// TIA Portal V19 export
FUNCTION_BLOCK "F_Zone05_FB"   // FB116, F_LAD
TITLE = SAFETY ZONE 07 - AREA 01 (PEELERS + STRAIGHTENER + JB + LOOP 1 FRONT)
// stored: Access Published
   VAR
      D04 : "Door_FB";
      D05 : "Door_FB";
      FNS : "ForceNormalStop";
      F_SafetyValve_CoilCar : "FDevice_Valve_FB";
      F_SafetyValve_Peeler : "FDevice_Valve_FB";
      F_SafetyValve_JB_Cut_Rest : "FDevice_Valve_FB";
      F_SafetyValve_JB_Cut_Work : "FDevice_Valve_FB";
      F_Contactor_HU_Area01_Motor : "FDevice_Contactor_FB";
      F_Sinamics_JBTorch : "FDevice_Sinamics_FB";
      F_Sinamics_JBPinchRoll : "FDevice_Sinamics_FB";
   END_VAR
   VAR_TEMP
      Fdbk : Bool;
   END_VAR
   VAR CONSTANT
      JB_TORCH_S120_STOPPING_TIME : Time := T#1s;
      JB_PINCHR_S120_STOPPING_TIME : Time := T#1s;
   END_VAR
BEGIN

REGION Network 1: < < < < < < < < < < DOOR > > > > > > > > > >
END_REGION

REGION Network 2: Zone Entry enable
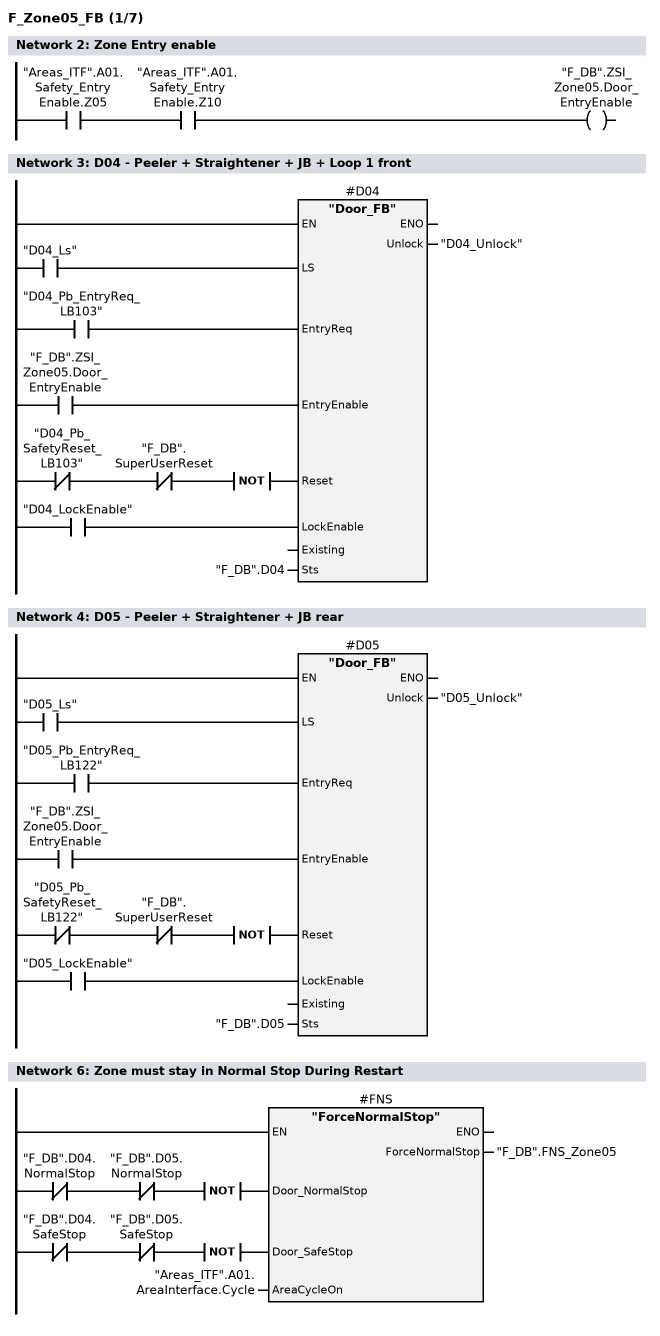
   RUNG wire#powerrail
      Contact( "Areas_ITF".A01.Safety_EntryEnable.Z05 )
      Contact( "Areas_ITF".A01.Safety_EntryEnable.Z10 )
      Coil( "F_DB".ZSI_Zone05.Door_EntryEnable )
   END_RUNG
   // the same network as SCL:
   "F_DB".ZSI_Zone05.Door_EntryEnable := "Areas_ITF".A01.Safety_EntryEnable.Z05 AND "Areas_ITF".A01.Safety_EntryEnable.Z10;
END_REGION

REGION Network 3: D04 - Peeler + Straightener + JB + Loop 1 front
   RUNG wire#powerrail
      #D04(LS := wire#w1, EntryReq := wire#w2, EntryEnable := wire#w3, Reset := wire#w4, LockEnable := wire#w5, Existing :=, Sts := "F_DB".D04, Unlock => "D04_Unlock")
   END_RUNG
   RUNG wire#powerrail
      Contact( "D04_Ls" )
   END_RUNG wire#w1
   RUNG wire#powerrail
      Contact( "D04_Pb_EntryReq_LB103" )
   END_RUNG wire#w2
   RUNG wire#powerrail
      Contact( "F_DB".ZSI_Zone05.Door_EntryEnable )
   END_RUNG wire#w3
   RUNG wire#powerrail
      I_Contact( "D04_Pb_SafetyReset_LB103" )
      I_Contact( "F_DB".SuperUserReset )
      Not()
   END_RUNG wire#w4
   RUNG wire#powerrail
      Contact( "D04_LockEnable" )
   END_RUNG wire#w5
   // the same network as SCL:
   #D04(LS := "D04_Ls",   // "Door_FB"
        EntryReq := "D04_Pb_EntryReq_LB103",
        EntryEnable := "F_DB".ZSI_Zone05.Door_EntryEnable,
        Reset := NOT (NOT "D04_Pb_SafetyReset_LB103" AND NOT "F_DB".SuperUserReset),
        LockEnable := "D04_LockEnable",
        Sts := "F_DB".D04,
        Unlock => "D04_Unlock");
END_REGION

REGION Network 4: D05 - Peeler + Straightener + JB rear
   RUNG wire#powerrail
      #D05(LS := wire#w1, EntryReq := wire#w2, EntryEnable := wire#w3, Reset := wire#w4, LockEnable := wire#w5, Existing :=, Sts := "F_DB".D05, Unlock => "D05_Unlock")
   END_RUNG
   RUNG wire#powerrail
      Contact( "D05_Ls" )
   END_RUNG wire#w1
   RUNG wire#powerrail
      Contact( "D05_Pb_EntryReq_LB122" )
   END_RUNG wire#w2
   RUNG wire#powerrail
      Contact( "F_DB".ZSI_Zone05.Door_EntryEnable )
   END_RUNG wire#w3
   RUNG wire#powerrail
      I_Contact( "D05_Pb_SafetyReset_LB122" )
      I_Contact( "F_DB".SuperUserReset )
      Not()
   END_RUNG wire#w4
   RUNG wire#powerrail
      Contact( "D05_LockEnable" )
   END_RUNG wire#w5
   // the same network as SCL:
   #D05(LS := "D05_Ls",   // "Door_FB"
        EntryReq := "D05_Pb_EntryReq_LB122",
        EntryEnable := "F_DB".ZSI_Zone05.Door_EntryEnable,
        Reset := NOT (NOT "D05_Pb_SafetyReset_LB122" AND NOT "F_DB".SuperUserReset),
        LockEnable := "D05_LockEnable",
        Sts := "F_DB".D05,
        Unlock => "D05_Unlock");
END_REGION

REGION Network 5: < < < < < < < < < < FORCE NORMAL STOP > > > > > > > > > >
END_REGION

REGION Network 6: Zone must stay in Normal Stop During Restart
   RUNG wire#powerrail
      #FNS(Door_NormalStop := wire#w1, Door_SafeStop := wire#w2, AreaCycleOn := "Areas_ITF".A01.AreaInterface.Cycle, ForceNormalStop => "F_DB".FNS_Zone05)
   END_RUNG
   RUNG wire#powerrail
      I_Contact( "F_DB".D04.NormalStop )
      I_Contact( "F_DB".D05.NormalStop )
      Not()
   END_RUNG wire#w1
   RUNG wire#powerrail
      I_Contact( "F_DB".D04.SafeStop )
      I_Contact( "F_DB".D05.SafeStop )
      Not()
   END_RUNG wire#w2
   // the same network as SCL:
   #FNS(Door_NormalStop := NOT (NOT "F_DB".D04.NormalStop AND NOT "F_DB".D05.NormalStop),   // "ForceNormalStop"
        Door_SafeStop := NOT (NOT "F_DB".D04.SafeStop AND NOT "F_DB".D05.SafeStop),
        AreaCycleOn := "Areas_ITF".A01.AreaInterface.Cycle,
        ForceNormalStop => "F_DB".FNS_Zone05);
END_REGION

REGION Network 7: < < < < < < < < < < ZONE SAFETY INTERFACE > > > > > > > > > >
END_REGION

REGION Network 8: Cumulative Zone Safety
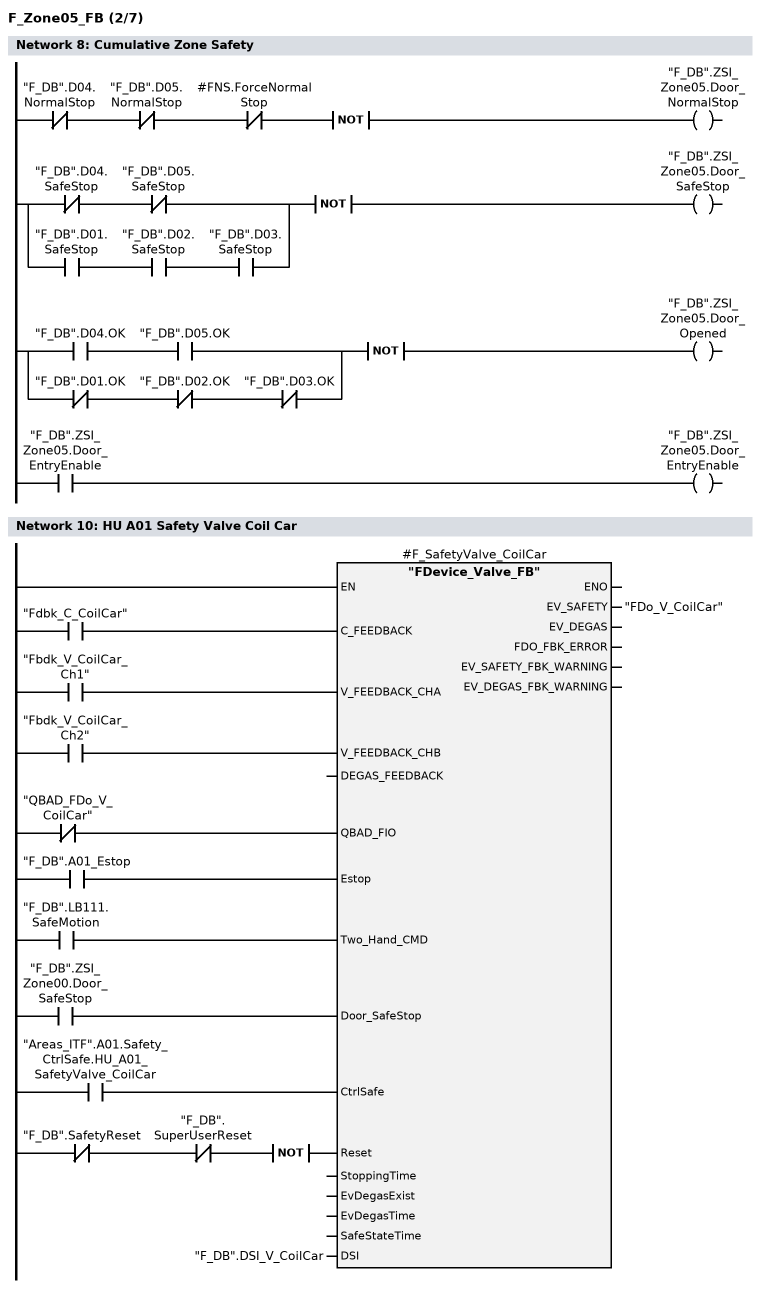
   RUNG wire#powerrail
      I_Contact( "F_DB".D04.NormalStop )
      I_Contact( "F_DB".D05.NormalStop )
      I_Contact( #FNS.ForceNormalStop )
      Not()
      Coil( "F_DB".ZSI_Zone05.Door_NormalStop )
   END_RUNG
   RUNG wire#powerrail
      I_Contact( "F_DB".D04.SafeStop )
      I_Contact( "F_DB".D05.SafeStop )
      wire#w1
      Not()
      Coil( "F_DB".ZSI_Zone05.Door_SafeStop )
   END_RUNG
   RUNG wire#powerrail
      Contact( "F_DB".D01.SafeStop )
      Contact( "F_DB".D02.SafeStop )
      Contact( "F_DB".D03.SafeStop )
   END_RUNG wire#w1
   RUNG wire#powerrail
      Contact( "F_DB".D04.OK )
      Contact( "F_DB".D05.OK )
      wire#w2
      Not()
      Coil( "F_DB".ZSI_Zone05.Door_Opened )
   END_RUNG
   RUNG wire#powerrail
      I_Contact( "F_DB".D01.OK )
      I_Contact( "F_DB".D02.OK )
      I_Contact( "F_DB".D03.OK )
   END_RUNG wire#w2
   RUNG wire#powerrail
      Contact( "F_DB".ZSI_Zone05.Door_EntryEnable )
      Coil( "F_DB".ZSI_Zone05.Door_EntryEnable )
   END_RUNG
   // the same network as SCL:
   "F_DB".ZSI_Zone05.Door_NormalStop := NOT (NOT "F_DB".D04.NormalStop AND NOT "F_DB".D05.NormalStop AND NOT #FNS.ForceNormalStop);
   "F_DB".ZSI_Zone05.Door_SafeStop := NOT ((NOT "F_DB".D04.SafeStop AND NOT "F_DB".D05.SafeStop) OR ("F_DB".D01.SafeStop AND "F_DB".D02.SafeStop AND "F_DB".D03.SafeStop));
   "F_DB".ZSI_Zone05.Door_Opened := NOT (("F_DB".D04.OK AND "F_DB".D05.OK) OR (NOT "F_DB".D01.OK AND NOT "F_DB".D02.OK AND NOT "F_DB".D03.OK));
   "F_DB".ZSI_Zone05.Door_EntryEnable := "F_DB".ZSI_Zone05.Door_EntryEnable;
END_REGION

REGION Network 9: < < < < < < < < < < DEVICES SAFETY VALVES > > > > > > > > > >
END_REGION

REGION Network 10: HU A01 Safety Valve Coil Car
   RUNG wire#powerrail
      #F_SafetyValve_CoilCar(C_FEEDBACK := wire#w1, V_FEEDBACK_CHA := wire#w2, V_FEEDBACK_CHB := wire#w3, QBAD_FIO := wire#w4, Estop := wire#w5, Two_Hand_CMD := wire#w6, Door_SafeStop := wire#w7, CtrlSafe := wire#w8, Reset := wire#w9, DEGAS_FEEDBACK :=, StoppingTime :=, EvDegasExist :=, EvDegasTime :=, SafeStateTime :=, DSI := "F_DB".DSI_V_CoilCar, EV_SAFETY => "FDo_V_CoilCar", EV_DEGAS =>, FDO_FBK_ERROR =>, EV_SAFETY_FBK_WARNING =>, EV_DEGAS_FBK_WARNING =>)
   END_RUNG
   RUNG wire#powerrail
      Contact( "Fdbk_C_CoilCar" )
   END_RUNG wire#w1
   RUNG wire#powerrail
      Contact( "Fbdk_V_CoilCar_Ch1" )
   END_RUNG wire#w2
   RUNG wire#powerrail
      Contact( "Fbdk_V_CoilCar_Ch2" )
   END_RUNG wire#w3
   RUNG wire#powerrail
      I_Contact( "QBAD_FDo_V_CoilCar" )
   END_RUNG wire#w4
   RUNG wire#powerrail
      Contact( "F_DB".A01_Estop )
   END_RUNG wire#w5
   RUNG wire#powerrail
      Contact( "F_DB".LB111.SafeMotion )
   END_RUNG wire#w6
   RUNG wire#powerrail
      Contact( "F_DB".ZSI_Zone00.Door_SafeStop )
   END_RUNG wire#w7
   RUNG wire#powerrail
      Contact( "Areas_ITF".A01.Safety_CtrlSafe.HU_A01_SafetyValve_CoilCar )
   END_RUNG wire#w8
   RUNG wire#powerrail
      I_Contact( "F_DB".SafetyReset )
      I_Contact( "F_DB".SuperUserReset )
      Not()
   END_RUNG wire#w9
   // the same network as SCL:
   #F_SafetyValve_CoilCar(C_FEEDBACK := "Fdbk_C_CoilCar",   // "FDevice_Valve_FB"
                          V_FEEDBACK_CHA := "Fbdk_V_CoilCar_Ch1",
                          V_FEEDBACK_CHB := "Fbdk_V_CoilCar_Ch2",
                          QBAD_FIO := NOT "QBAD_FDo_V_CoilCar",
                          Estop := "F_DB".A01_Estop,
                          Two_Hand_CMD := "F_DB".LB111.SafeMotion,
                          Door_SafeStop := "F_DB".ZSI_Zone00.Door_SafeStop,
                          CtrlSafe := "Areas_ITF".A01.Safety_CtrlSafe.HU_A01_SafetyValve_CoilCar,
                          Reset := NOT (NOT "F_DB".SafetyReset AND NOT "F_DB".SuperUserReset),
                          DSI := "F_DB".DSI_V_CoilCar,
                          EV_SAFETY => "FDo_V_CoilCar");
END_REGION

REGION Network 11: HU A01 Safety Valve Peeler
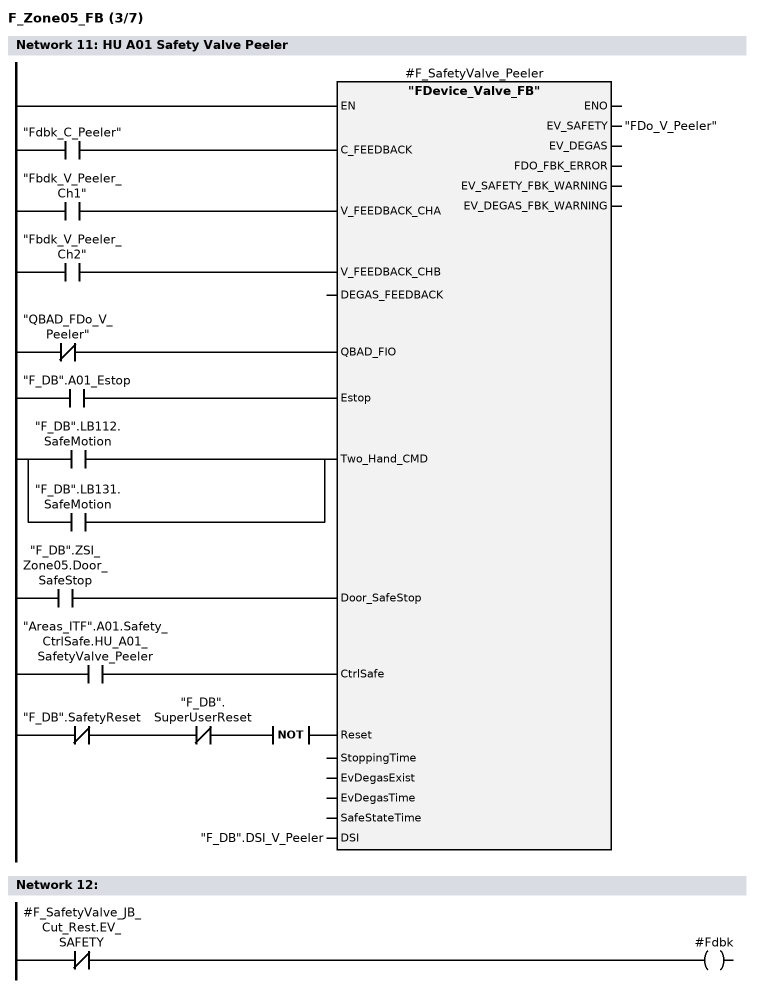
   RUNG wire#powerrail
      #F_SafetyValve_Peeler(C_FEEDBACK := wire#w1, V_FEEDBACK_CHA := wire#w2, V_FEEDBACK_CHB := wire#w3, QBAD_FIO := wire#w4, Estop := wire#w5, Two_Hand_CMD := wire#w6, Door_SafeStop := wire#w7, CtrlSafe := wire#w8, Reset := wire#w9, DEGAS_FEEDBACK :=, StoppingTime :=, EvDegasExist :=, EvDegasTime :=, SafeStateTime :=, DSI := "F_DB".DSI_V_Peeler, EV_SAFETY => "FDo_V_Peeler", EV_DEGAS =>, FDO_FBK_ERROR =>, EV_SAFETY_FBK_WARNING =>, EV_DEGAS_FBK_WARNING =>)
   END_RUNG
   RUNG wire#powerrail
      Contact( "Fdbk_C_Peeler" )
   END_RUNG wire#w1
   RUNG wire#powerrail
      Contact( "Fbdk_V_Peeler_Ch1" )
   END_RUNG wire#w2
   RUNG wire#powerrail
      Contact( "Fbdk_V_Peeler_Ch2" )
   END_RUNG wire#w3
   RUNG wire#powerrail
      I_Contact( "QBAD_FDo_V_Peeler" )
   END_RUNG wire#w4
   RUNG wire#powerrail
      Contact( "F_DB".A01_Estop )
   END_RUNG wire#w5
   RUNG wire#powerrail
      Contact( "F_DB".LB112.SafeMotion )
   END_RUNG wire#w6
   RUNG wire#powerrail
      Contact( "F_DB".LB131.SafeMotion )
   END_RUNG wire#w6
   RUNG wire#powerrail
      Contact( "F_DB".ZSI_Zone05.Door_SafeStop )
   END_RUNG wire#w7
   RUNG wire#powerrail
      Contact( "Areas_ITF".A01.Safety_CtrlSafe.HU_A01_SafetyValve_Peeler )
   END_RUNG wire#w8
   RUNG wire#powerrail
      I_Contact( "F_DB".SafetyReset )
      I_Contact( "F_DB".SuperUserReset )
      Not()
   END_RUNG wire#w9
   // the same network as SCL:
   #F_SafetyValve_Peeler(C_FEEDBACK := "Fdbk_C_Peeler",   // "FDevice_Valve_FB"
                         V_FEEDBACK_CHA := "Fbdk_V_Peeler_Ch1",
                         V_FEEDBACK_CHB := "Fbdk_V_Peeler_Ch2",
                         QBAD_FIO := NOT "QBAD_FDo_V_Peeler",
                         Estop := "F_DB".A01_Estop,
                         Two_Hand_CMD := "F_DB".LB112.SafeMotion OR "F_DB".LB131.SafeMotion,
                         Door_SafeStop := "F_DB".ZSI_Zone05.Door_SafeStop,
                         CtrlSafe := "Areas_ITF".A01.Safety_CtrlSafe.HU_A01_SafetyValve_Peeler,
                         Reset := NOT (NOT "F_DB".SafetyReset AND NOT "F_DB".SuperUserReset),
                         DSI := "F_DB".DSI_V_Peeler,
                         EV_SAFETY => "FDo_V_Peeler");
END_REGION

REGION Network 12
   RUNG wire#powerrail
      I_Contact( #F_SafetyValve_JB_Cut_Rest.EV_SAFETY )
      Coil( #Fdbk )
   END_RUNG
   // the same network as SCL:
   #Fdbk := NOT #F_SafetyValve_JB_Cut_Rest.EV_SAFETY;
END_REGION

REGION Network 13: HU A01 Safety Valve JB Cut Rest
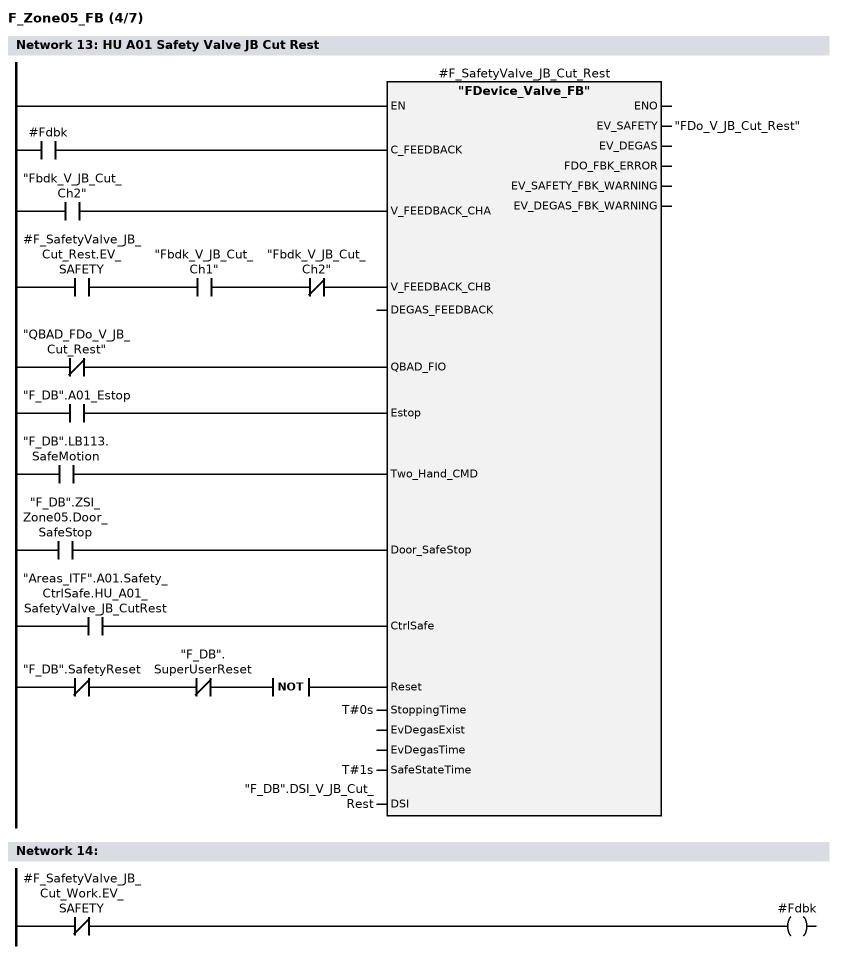
   RUNG wire#powerrail
      #F_SafetyValve_JB_Cut_Rest(C_FEEDBACK := wire#w1, V_FEEDBACK_CHA := wire#w2, V_FEEDBACK_CHB := wire#w3, QBAD_FIO := wire#w4, Estop := wire#w5, Two_Hand_CMD := wire#w6, Door_SafeStop := wire#w7, CtrlSafe := wire#w8, Reset := wire#w9, DEGAS_FEEDBACK :=, StoppingTime := T#0s, EvDegasExist :=, EvDegasTime :=, SafeStateTime := T#1s, DSI := "F_DB".DSI_V_JB_Cut_Rest, EV_SAFETY => "FDo_V_JB_Cut_Rest", EV_DEGAS =>, FDO_FBK_ERROR =>, EV_SAFETY_FBK_WARNING =>, EV_DEGAS_FBK_WARNING =>)
   END_RUNG
   RUNG wire#powerrail
      Contact( #Fdbk )
   END_RUNG wire#w1
   RUNG wire#powerrail
      Contact( "Fbdk_V_JB_Cut_Ch2" )
   END_RUNG wire#w2
   RUNG wire#powerrail
      Contact( #F_SafetyValve_JB_Cut_Rest.EV_SAFETY )
      Contact( "Fbdk_V_JB_Cut_Ch1" )
      I_Contact( "Fbdk_V_JB_Cut_Ch2" )
   END_RUNG wire#w3
   RUNG wire#powerrail
      I_Contact( "QBAD_FDo_V_JB_Cut_Rest" )
   END_RUNG wire#w4
   RUNG wire#powerrail
      Contact( "F_DB".A01_Estop )
   END_RUNG wire#w5
   RUNG wire#powerrail
      Contact( "F_DB".LB113.SafeMotion )
   END_RUNG wire#w6
   RUNG wire#powerrail
      Contact( "F_DB".ZSI_Zone05.Door_SafeStop )
   END_RUNG wire#w7
   RUNG wire#powerrail
      Contact( "Areas_ITF".A01.Safety_CtrlSafe.HU_A01_SafetyValve_JB_CutRest )
   END_RUNG wire#w8
   RUNG wire#powerrail
      I_Contact( "F_DB".SafetyReset )
      I_Contact( "F_DB".SuperUserReset )
      Not()
   END_RUNG wire#w9
   // the same network as SCL:
   #F_SafetyValve_JB_Cut_Rest(C_FEEDBACK := #Fdbk,   // "FDevice_Valve_FB"
                           V_FEEDBACK_CHA := "Fbdk_V_JB_Cut_Ch2",
                           V_FEEDBACK_CHB := #F_SafetyValve_JB_Cut_Rest.EV_SAFETY AND "Fbdk_V_JB_Cut_Ch1" AND NOT "Fbdk_V_JB_Cut_Ch2",
                           QBAD_FIO := NOT "QBAD_FDo_V_JB_Cut_Rest",
                           Estop := "F_DB".A01_Estop,
                           Two_Hand_CMD := "F_DB".LB113.SafeMotion,
                           Door_SafeStop := "F_DB".ZSI_Zone05.Door_SafeStop,
                           CtrlSafe := "Areas_ITF".A01.Safety_CtrlSafe.HU_A01_SafetyValve_JB_CutRest,
                           Reset := NOT (NOT "F_DB".SafetyReset AND NOT "F_DB".SuperUserReset),
                           StoppingTime := T#0s,
                           SafeStateTime := T#1s,
                           DSI := "F_DB".DSI_V_JB_Cut_Rest,
                           EV_SAFETY => "FDo_V_JB_Cut_Rest");
END_REGION

REGION Network 14
   RUNG wire#powerrail
      I_Contact( #F_SafetyValve_JB_Cut_Work.EV_SAFETY )
      Coil( #Fdbk )
   END_RUNG
   // the same network as SCL:
   #Fdbk := NOT #F_SafetyValve_JB_Cut_Work.EV_SAFETY;
END_REGION

REGION Network 15: HU A01 Safety Valve JB Cut Work
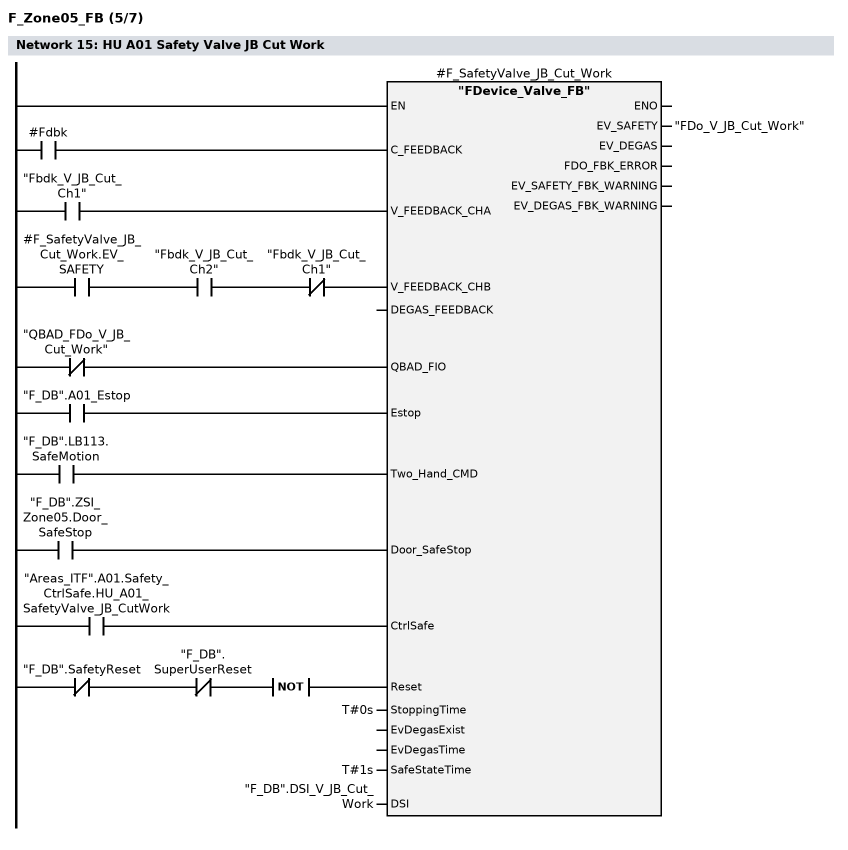
   RUNG wire#powerrail
      #F_SafetyValve_JB_Cut_Work(C_FEEDBACK := wire#w1, V_FEEDBACK_CHA := wire#w2, V_FEEDBACK_CHB := wire#w3, QBAD_FIO := wire#w4, Estop := wire#w5, Two_Hand_CMD := wire#w6, Door_SafeStop := wire#w7, CtrlSafe := wire#w8, Reset := wire#w9, DEGAS_FEEDBACK :=, StoppingTime := T#0s, EvDegasExist :=, EvDegasTime :=, SafeStateTime := T#1s, DSI := "F_DB".DSI_V_JB_Cut_Work, EV_SAFETY => "FDo_V_JB_Cut_Work", EV_DEGAS =>, FDO_FBK_ERROR =>, EV_SAFETY_FBK_WARNING =>, EV_DEGAS_FBK_WARNING =>)
   END_RUNG
   RUNG wire#powerrail
      Contact( #Fdbk )
   END_RUNG wire#w1
   RUNG wire#powerrail
      Contact( "Fbdk_V_JB_Cut_Ch1" )
   END_RUNG wire#w2
   RUNG wire#powerrail
      Contact( #F_SafetyValve_JB_Cut_Work.EV_SAFETY )
      Contact( "Fbdk_V_JB_Cut_Ch2" )
      I_Contact( "Fbdk_V_JB_Cut_Ch1" )
   END_RUNG wire#w3
   RUNG wire#powerrail
      I_Contact( "QBAD_FDo_V_JB_Cut_Work" )
   END_RUNG wire#w4
   RUNG wire#powerrail
      Contact( "F_DB".A01_Estop )
   END_RUNG wire#w5
   RUNG wire#powerrail
      Contact( "F_DB".LB113.SafeMotion )
   END_RUNG wire#w6
   RUNG wire#powerrail
      Contact( "F_DB".ZSI_Zone05.Door_SafeStop )
   END_RUNG wire#w7
   RUNG wire#powerrail
      Contact( "Areas_ITF".A01.Safety_CtrlSafe.HU_A01_SafetyValve_JB_CutWork )
   END_RUNG wire#w8
   RUNG wire#powerrail
      I_Contact( "F_DB".SafetyReset )
      I_Contact( "F_DB".SuperUserReset )
      Not()
   END_RUNG wire#w9
   // the same network as SCL:
   #F_SafetyValve_JB_Cut_Work(C_FEEDBACK := #Fdbk,   // "FDevice_Valve_FB"
                           V_FEEDBACK_CHA := "Fbdk_V_JB_Cut_Ch1",
                           V_FEEDBACK_CHB := #F_SafetyValve_JB_Cut_Work.EV_SAFETY AND "Fbdk_V_JB_Cut_Ch2" AND NOT "Fbdk_V_JB_Cut_Ch1",
                           QBAD_FIO := NOT "QBAD_FDo_V_JB_Cut_Work",
                           Estop := "F_DB".A01_Estop,
                           Two_Hand_CMD := "F_DB".LB113.SafeMotion,
                           Door_SafeStop := "F_DB".ZSI_Zone05.Door_SafeStop,
                           CtrlSafe := "Areas_ITF".A01.Safety_CtrlSafe.HU_A01_SafetyValve_JB_CutWork,
                           Reset := NOT (NOT "F_DB".SafetyReset AND NOT "F_DB".SuperUserReset),
                           StoppingTime := T#0s,
                           SafeStateTime := T#1s,
                           DSI := "F_DB".DSI_V_JB_Cut_Work,
                           EV_SAFETY => "FDo_V_JB_Cut_Work");
END_REGION

REGION Network 16: >
END_REGION

REGION Network 17: < < < < < < < < < < DEVICES CONTACTORS > > > > > > > > > >
END_REGION

REGION Network 18: HU A01 Motor contactor
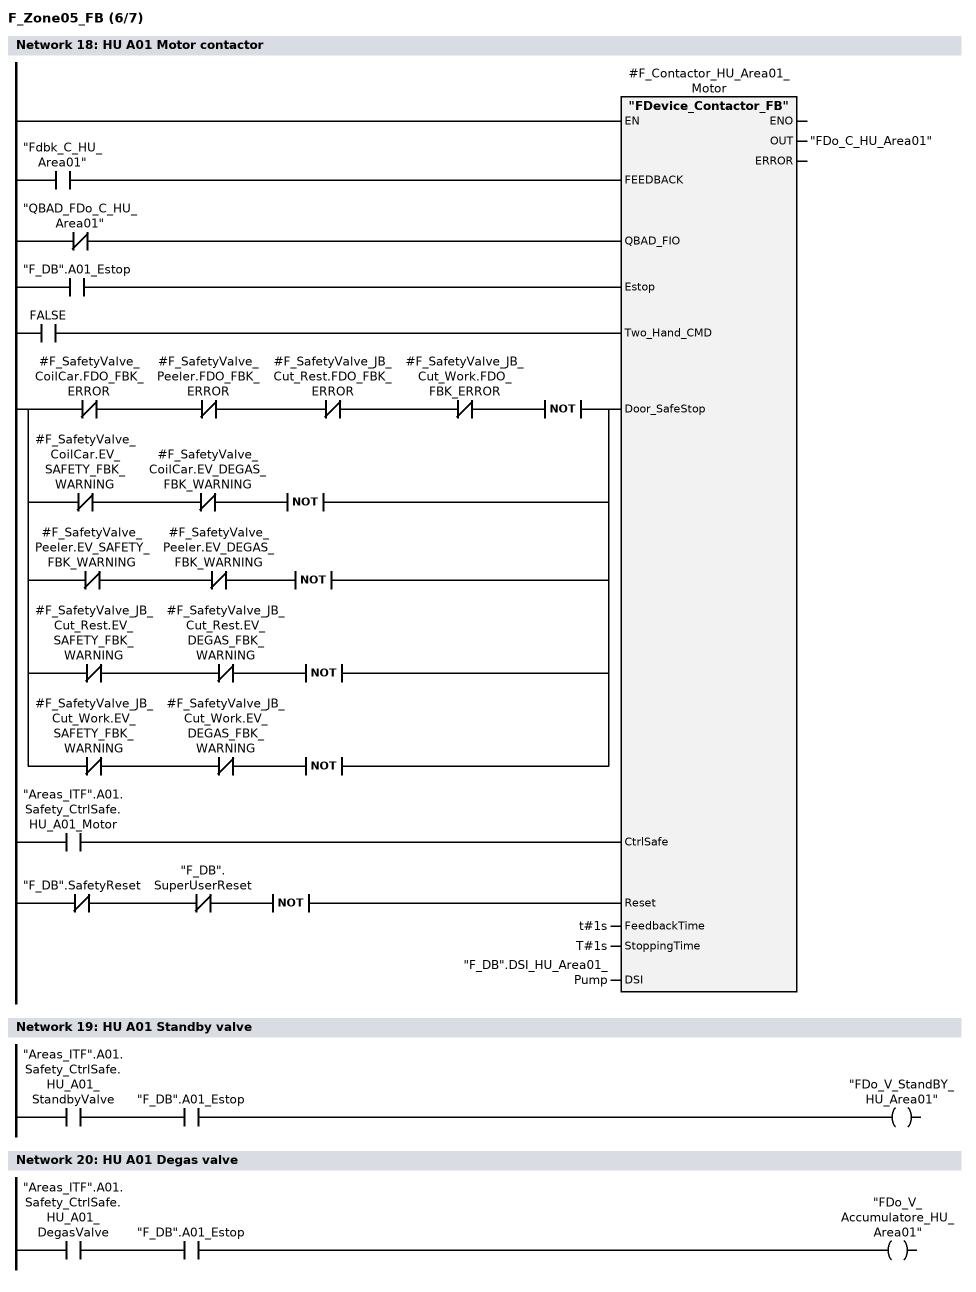
   RUNG wire#powerrail
      #F_Contactor_HU_Area01_Motor(FEEDBACK := wire#w1, QBAD_FIO := wire#w2, Estop := wire#w3, Two_Hand_CMD := wire#w4, Door_SafeStop := wire#w5, CtrlSafe := wire#w6, Reset := wire#w7, FeedbackTime := t#1s, StoppingTime := T#1s, DSI := "F_DB".DSI_HU_Area01_Pump, OUT => "FDo_C_HU_Area01", ERROR =>)
   END_RUNG
   RUNG wire#powerrail
      Contact( "Fdbk_C_HU_Area01" )
   END_RUNG wire#w1
   RUNG wire#powerrail
      I_Contact( "QBAD_FDo_C_HU_Area01" )
   END_RUNG wire#w2
   RUNG wire#powerrail
      Contact( "F_DB".A01_Estop )
   END_RUNG wire#w3
   RUNG wire#powerrail
      Contact( FALSE )
   END_RUNG wire#w4
   RUNG wire#powerrail
      I_Contact( #F_SafetyValve_CoilCar.FDO_FBK_ERROR )
      I_Contact( #F_SafetyValve_Peeler.FDO_FBK_ERROR )
      I_Contact( #F_SafetyValve_JB_Cut_Rest.FDO_FBK_ERROR )
      I_Contact( #F_SafetyValve_JB_Cut_Work.FDO_FBK_ERROR )
      Not()
   END_RUNG wire#w5
   RUNG wire#powerrail
      I_Contact( #F_SafetyValve_CoilCar.EV_SAFETY_FBK_WARNING )
      I_Contact( #F_SafetyValve_CoilCar.EV_DEGAS_FBK_WARNING )
      Not()
   END_RUNG wire#w5
   RUNG wire#powerrail
      I_Contact( #F_SafetyValve_Peeler.EV_SAFETY_FBK_WARNING )
      I_Contact( #F_SafetyValve_Peeler.EV_DEGAS_FBK_WARNING )
      Not()
   END_RUNG wire#w5
   RUNG wire#powerrail
      I_Contact( #F_SafetyValve_JB_Cut_Rest.EV_SAFETY_FBK_WARNING )
      I_Contact( #F_SafetyValve_JB_Cut_Rest.EV_DEGAS_FBK_WARNING )
      Not()
   END_RUNG wire#w5
   RUNG wire#powerrail
      I_Contact( #F_SafetyValve_JB_Cut_Work.EV_SAFETY_FBK_WARNING )
      I_Contact( #F_SafetyValve_JB_Cut_Work.EV_DEGAS_FBK_WARNING )
      Not()
   END_RUNG wire#w5
   RUNG wire#powerrail
      Contact( "Areas_ITF".A01.Safety_CtrlSafe.HU_A01_Motor )
   END_RUNG wire#w6
   RUNG wire#powerrail
      I_Contact( "F_DB".SafetyReset )
      I_Contact( "F_DB".SuperUserReset )
      Not()
   END_RUNG wire#w7
   // the same network as SCL:
   #F_Contactor_HU_Area01_Motor(FEEDBACK := "Fdbk_C_HU_Area01",   // "FDevice_Contactor_FB"
                           QBAD_FIO := NOT "QBAD_FDo_C_HU_Area01",
                           Estop := "F_DB".A01_Estop,
                           Two_Hand_CMD := FALSE,
                           Door_SafeStop := NOT (NOT #F_SafetyValve_CoilCar.FDO_FBK_ERROR AND NOT #F_SafetyValve_Peeler.FDO_FBK_ERROR AND NOT #F_SafetyValve_JB_Cut_Rest.FDO_FBK_ERROR AND NOT #F_SafetyValve_JB_Cut_Work.FDO_FBK_ERROR) OR NOT (NOT #F_SafetyValve_CoilCar.EV_SAFETY_FBK_WARNING AND NOT #F_SafetyValve_CoilCar.EV_DEGAS_FBK_WARNING) OR NOT (NOT #F_SafetyValve_Peeler.EV_SAFETY_FBK_WARNING AND NOT #F_SafetyValve_Peeler.EV_DEGAS_FBK_WARNING) OR NOT (NOT #F_SafetyValve_JB_Cut_Rest.EV_SAFETY_FBK_WARNING AND NOT #F_SafetyValve_JB_Cut_Rest.EV_DEGAS_FBK_WARNING) OR NOT (NOT #F_SafetyValve_JB_Cut_Work.EV_SAFETY_FBK_WARNING AND NOT #F_SafetyValve_JB_Cut_Work.EV_DEGAS_FBK_WARNING),
                           CtrlSafe := "Areas_ITF".A01.Safety_CtrlSafe.HU_A01_Motor,
                           Reset := NOT (NOT "F_DB".SafetyReset AND NOT "F_DB".SuperUserReset),
                           FeedbackTime := t#1s,
                           StoppingTime := T#1s,
                           DSI := "F_DB".DSI_HU_Area01_Pump,
                           OUT => "FDo_C_HU_Area01");
END_REGION

REGION Network 19: HU A01 Standby valve
   RUNG wire#powerrail
      Contact( "Areas_ITF".A01.Safety_CtrlSafe.HU_A01_StandbyValve )
      Contact( "F_DB".A01_Estop )
      Coil( "FDo_V_StandBY_HU_Area01" )
   END_RUNG
   // the same network as SCL:
   "FDo_V_StandBY_HU_Area01" := "Areas_ITF".A01.Safety_CtrlSafe.HU_A01_StandbyValve AND "F_DB".A01_Estop;
END_REGION

REGION Network 20: HU A01 Degas valve
   RUNG wire#powerrail
      Contact( "Areas_ITF".A01.Safety_CtrlSafe.HU_A01_DegasValve )
      Contact( "F_DB".A01_Estop )
      Coil( "FDo_V_Accumulatore_HU_Area01" )
   END_RUNG
   // the same network as SCL:
   "FDo_V_Accumulatore_HU_Area01" := "Areas_ITF".A01.Safety_CtrlSafe.HU_A01_DegasValve AND "F_DB".A01_Estop;
END_REGION

REGION Network 21: >
END_REGION

REGION Network 22: < < < < < < < < < < DEVICES S120 > > > > > > > > > >
END_REGION

REGION Network 23: S120 - JB Welder Torch
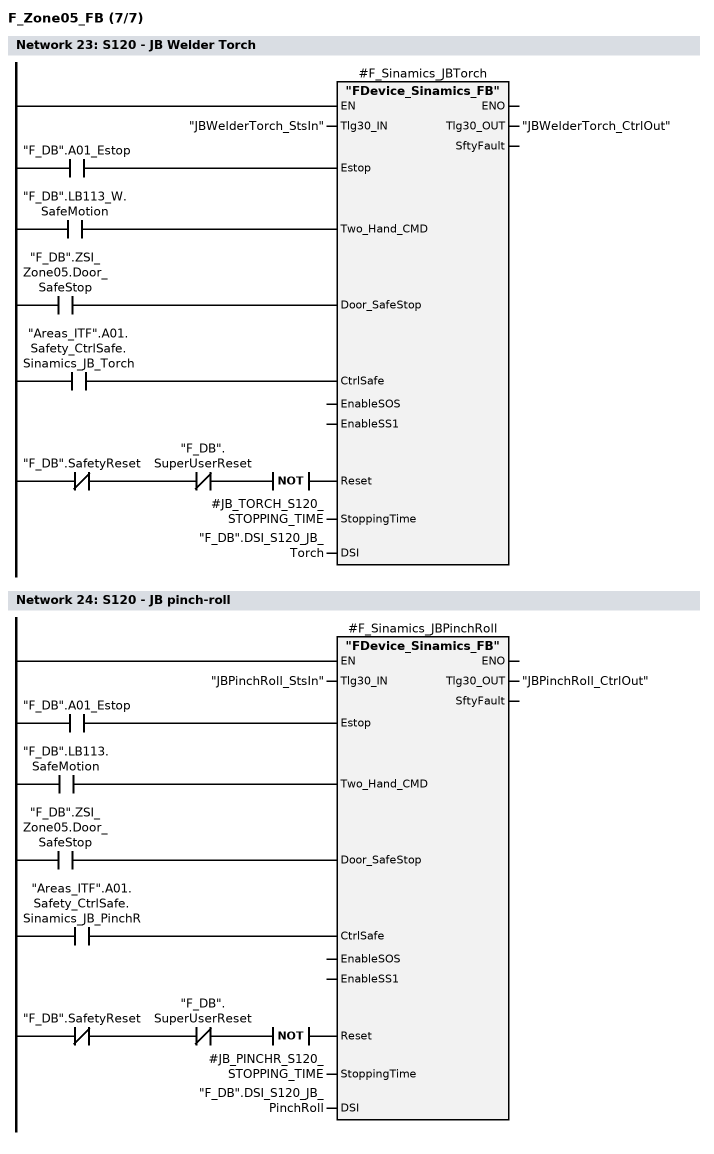
   RUNG wire#powerrail
      #F_Sinamics_JBTorch(Estop := wire#w1, Two_Hand_CMD := wire#w2, Door_SafeStop := wire#w3, CtrlSafe := wire#w4, Reset := wire#w5, Tlg30_IN := "JBWelderTorch_StsIn", EnableSOS :=, EnableSS1 :=, StoppingTime := #JB_TORCH_S120_STOPPING_TIME, DSI := "F_DB".DSI_S120_JB_Torch, Tlg30_OUT => "JBWelderTorch_CtrlOut", SftyFault =>)
   END_RUNG
   RUNG wire#powerrail
      Contact( "F_DB".A01_Estop )
   END_RUNG wire#w1
   RUNG wire#powerrail
      Contact( "F_DB".LB113_W.SafeMotion )
   END_RUNG wire#w2
   RUNG wire#powerrail
      Contact( "F_DB".ZSI_Zone05.Door_SafeStop )
   END_RUNG wire#w3
   RUNG wire#powerrail
      Contact( "Areas_ITF".A01.Safety_CtrlSafe.Sinamics_JB_Torch )
   END_RUNG wire#w4
   RUNG wire#powerrail
      I_Contact( "F_DB".SafetyReset )
      I_Contact( "F_DB".SuperUserReset )
      Not()
   END_RUNG wire#w5
   // the same network as SCL:
   #F_Sinamics_JBTorch(Tlg30_IN := "JBWelderTorch_StsIn",   // "FDevice_Sinamics_FB"
                       Estop := "F_DB".A01_Estop,
                       Two_Hand_CMD := "F_DB".LB113_W.SafeMotion,
                       Door_SafeStop := "F_DB".ZSI_Zone05.Door_SafeStop,
                       CtrlSafe := "Areas_ITF".A01.Safety_CtrlSafe.Sinamics_JB_Torch,
                       Reset := NOT (NOT "F_DB".SafetyReset AND NOT "F_DB".SuperUserReset),
                       StoppingTime := #JB_TORCH_S120_STOPPING_TIME,
                       DSI := "F_DB".DSI_S120_JB_Torch,
                       Tlg30_OUT => "JBWelderTorch_CtrlOut");
END_REGION

REGION Network 24: S120 - JB pinch-roll
   RUNG wire#powerrail
      #F_Sinamics_JBPinchRoll(Estop := wire#w1, Two_Hand_CMD := wire#w2, Door_SafeStop := wire#w3, CtrlSafe := wire#w4, Reset := wire#w5, Tlg30_IN := "JBPinchRoll_StsIn", EnableSOS :=, EnableSS1 :=, StoppingTime := #JB_PINCHR_S120_STOPPING_TIME, DSI := "F_DB".DSI_S120_JB_PinchRoll, Tlg30_OUT => "JBPinchRoll_CtrlOut", SftyFault =>)
   END_RUNG
   RUNG wire#powerrail
      Contact( "F_DB".A01_Estop )
   END_RUNG wire#w1
   RUNG wire#powerrail
      Contact( "F_DB".LB113.SafeMotion )
   END_RUNG wire#w2
   RUNG wire#powerrail
      Contact( "F_DB".ZSI_Zone05.Door_SafeStop )
   END_RUNG wire#w3
   RUNG wire#powerrail
      Contact( "Areas_ITF".A01.Safety_CtrlSafe.Sinamics_JB_PinchR )
   END_RUNG wire#w4
   RUNG wire#powerrail
      I_Contact( "F_DB".SafetyReset )
      I_Contact( "F_DB".SuperUserReset )
      Not()
   END_RUNG wire#w5
   // the same network as SCL:
   #F_Sinamics_JBPinchRoll(Tlg30_IN := "JBPinchRoll_StsIn",   // "FDevice_Sinamics_FB"
                           Estop := "F_DB".A01_Estop,
                           Two_Hand_CMD := "F_DB".LB113.SafeMotion,
                           Door_SafeStop := "F_DB".ZSI_Zone05.Door_SafeStop,
                           CtrlSafe := "Areas_ITF".A01.Safety_CtrlSafe.Sinamics_JB_PinchR,
                           Reset := NOT (NOT "F_DB".SafetyReset AND NOT "F_DB".SuperUserReset),
                           StoppingTime := #JB_PINCHR_S120_STOPPING_TIME,
                           DSI := "F_DB".DSI_S120_JB_PinchRoll,
                           Tlg30_OUT => "JBPinchRoll_CtrlOut");
END_REGION

REGION Network 25: >
END_REGION

REGION Network 26: >
END_REGION

REGION Network 27: >
END_REGION
END_FUNCTION_BLOCK
